TYPE ST_ValveError :
STRUCT 
	errOpenTimeout: 		STRING	:= 'alarm open timeout';
	errLostOpenPosition: 	STRING	:= 'lost open position';
	errCloseTimeout: 		STRING	:= 'alarm closing timeout';
	errLostClosePosition: 	STRING	:= 'lost close position';
	errBothSensorOn: 		STRING	:= 'alarm both sensor on';
	warnRequestAuto:		STRING	:= 'request auto control from parent em';
END_STRUCT
END_TYPE

(* stored: Version 1.1.0.1, ProductVersion 3.1.4024.13
   DUT ST_ValveError: Id {16a7da1a-b268-4d73-948a-5454623bf3a2} *)
